ORGANIZATION_BLOCK "Main"
TITLE = "Main Program Sweep (Cycle)"
{ S7_Optimized_Access := 'TRUE' }
VERSION : 0.1

BEGIN
	// Call test FC for pointer datatypes
	"FC_TestCallPointers"();
END_ORGANIZATION_BLOCK

